FUNCTION_BLOCK FB_09_SetOverridePercent
VAR_INPUT
	OverridePercent:LREAL:=100;
END_VAR
VAR_OUTPUT
END_VAR
VAR_IN_OUT
	stItpToPlc :NCTOPLC_NCICHANNEL_REF;
	stPlcToItp:PLCTONC_NCICHANNEL_REF;
END_VAR
VAR
END_VAR

ItpSetOverridePercent(fOverridePercent:= OverridePercent, sPlcToNci:= stPlcToItp);

END_FUNCTION_BLOCK

(* stored: Version 1.1.0.1, ProductVersion 3.1.4024.12
   POU FB_09_SetOverridePercent: Id {a5f0b5d6-267b-4859-859f-f9845fd1058b}, SpecialFunc None *)
